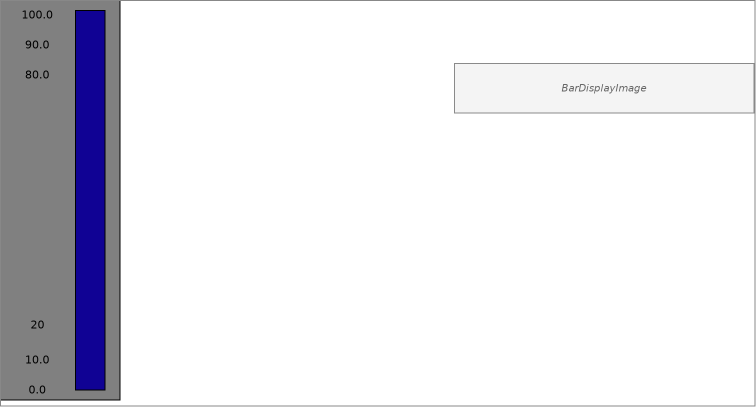
VISUALIZATION visu  // 756x407
    BarDisplayImage (454,63 300x50), style: BarDisplayImage-Gray, scale format: %.1f, scale 0..100
    Rectangle (0,0 120x400)
    Rectangle (75,10 30x380)
    Label (0,375 75x30), "0.0"
    Label (0,0 75x30), "100.0"
    Label (0,30 75x30), "90.0"
    Label (0,60 75x30), "80.0"
    Label (0,345 75x30), "10.0"
    Label (0,310 75x30), "20"
END_VISUALIZATION

(* stored: Version 1.1.0.1, ProductVersion 3.1.4022.17
   Visu visu: Id {06898ce8-f314-418c-bb91-9f31da0da354} *)
